# EPICS SNL sequencer program: siteApps/Helium_Inventory-1-0/inventoryApp/src/sncMakeTotalInventory.stt
program sncMakeTotalInventory

option +r;

double massflows[95];
assign massflows to {
	"SCL31-BL01:CM01-LT8401:MassFlow", "SCL31-BL01:CM02-LT8401:MassFlow", "SCL31-BL01:CM03-LT8401:MassFlow", "SCL31-BL01:CM04-LT8401:MassFlow", "SCL31-BL01:CM05-LT8401:MassFlow",
	"SCL31-BL01:CM06-LT8401:MassFlow", "SCL31-BL01:CM07-LT8401:MassFlow", "SCL31-BL01:CM08-LT8401:MassFlow", "SCL31-BL01:CM09-LT8401:MassFlow", "SCL31-BL01:CM10-LT8401:MassFlow",
	"SCL31-BL01:CM11-LT8401:MassFlow", "SCL31-BL01:CM12-LT8401:MassFlow", "SCL31-BL01:CM13-LT8401:MassFlow", "SCL31-BL01:CM14-LT8401:MassFlow", "SCL31-BL01:CM15-LT8401:MassFlow",
	"SCL31-BL01:CM16-LT8401:MassFlow", "SCL31-BL01:CM17-LT8401:MassFlow", "SCL31-BL01:CM18-LT8401:MassFlow", "SCL31-BL01:CM19-LT8401:MassFlow", "SCL31-BL01:CM20-LT8401:MassFlow",
	"SCL31-BL01:CM21-LT8401:MassFlow", "SCL31-BL01:CM22-LT8401:MassFlow", "SCL32-BL02:CM01-LT8401:MassFlow", "SCL32-BL02:CM02-LT8401:MassFlow", "SCL32-BL02:CM03-LT8401:MassFlow",
	"SCL32-BL02:CM04-LT8401:MassFlow", "SCL32-BL02:CM05-LT8401:MassFlow", "SCL32-BL02:CM06-LT8401:MassFlow", "SCL32-BL02:CM07-LT8401:MassFlow", "SCL32-BL02:CM08-LT8401:MassFlow",
	"SCL32-BL02:CM09-LT8401:MassFlow", "SCL32-BL02:CM10-LT8401:MassFlow", "SCL32-BL02:CM11-LT8401:MassFlow", "SCL32-BL02:CM12-LT8401:MassFlow", "SCL32-BL02:CM13-LT8401:MassFlow",
	"P2DT-BL04:CM01-LT8401:MassFlow", "SCL32-BL03:CM01-LT8401:MassFlow", "SCL32-BL03:CM02-LT8401:MassFlow", "SCL32-BL03:CM03-LT8401:MassFlow", "SCL32-BL03:CM04-LT8401:MassFlow",
	"SCL32-BL03:CM05-LT8401:MassFlow", "SCL32-BL03:CM06-LT8401:MassFlow", "SCL32-BL03:CM07-LT8401:MassFlow", "SCL32-BL03:CM08-LT8401:MassFlow", "SCL32-BL03:CM09-LT8401:MassFlow",
	"SCL32-BL03:CM10-LT8401:MassFlow", "SCL32-BL03:CM11-LT8401:MassFlow", "SCL32-BL03:CM12-LT8401:MassFlow", "SCL32-BL03:CM13-LT8401:MassFlow", "SCL32-BL03:CM14-LT8401:MassFlow",
	"SCL32-BL03:CM15-LT8401:MassFlow", "SCL32-BL03:CM16-LT8401:MassFlow", "SCL32-BL03:CM17-LT8401:MassFlow", "SCL32-BL03:CM18-LT8401:MassFlow", "SCL32-BL03:CM19-LT8401:MassFlow",
	"SCL32-BL02:CM01-LT8201:MassFlow", "SCL32-BL02:CM02-LT8201:MassFlow", "SCL32-BL02:CM03-LT8201:MassFlow", "SCL32-BL02:CM04-LT8201:MassFlow", "SCL32-BL02:CM05-LT8201:MassFlow",
	"SCL32-BL02:CM06-LT8201:MassFlow", "SCL32-BL02:CM07-LT8201:MassFlow", "SCL32-BL02:CM08-LT8201:MassFlow", "SCL32-BL02:CM09-LT8201:MassFlow", "SCL32-BL02:CM10-LT8201:MassFlow",
	"SCL32-BL02:CM11-LT8201:MassFlow", "SCL32-BL02:CM12-LT8201:MassFlow", "SCL32-BL02:CM13-LT8201:MassFlow", "P2DT-BL04:CM01-LT8201:MassFlow", "SCL32-BL03:CM01-LT8201:MassFlow",
	"SCL32-BL03:CM02-LT8201:MassFlow", "SCL32-BL03:CM03-LT8201:MassFlow", "SCL32-BL03:CM04-LT8201:MassFlow", "SCL32-BL03:CM05-LT8201:MassFlow", "SCL32-BL03:CM06-LT8201:MassFlow",
	"SCL32-BL03:CM07-LT8201:MassFlow", "SCL32-BL03:CM08-LT8201:MassFlow", "SCL32-BL03:CM09-LT8201:MassFlow", "SCL32-BL03:CM10-LT8201:MassFlow", "SCL32-BL03:CM11-LT8201:MassFlow",
	"SCL32-BL03:CM12-LT8201:MassFlow", "SCL32-BL03:CM13-LT8201:MassFlow", "SCL32-BL03:CM14-LT8201:MassFlow", "SCL32-BL03:CM15-LT8201:MassFlow", "SCL32-BL03:CM16-LT8201:MassFlow",
	"SCL32-BL03:CM17-LT8201:MassFlow", "SCL32-BL03:CM18-LT8201:MassFlow", "SCL32-BL03:CM19-LT8201:MassFlow", "Cryo-CDL00:TBx01-LT8401:2KReturn", "Cryo-CDL00:TBx01-LT8401:2KSupply",
	"Cryo-CDL00:TBx01-LT8401:4KReturn", "Cryo-CDL00:TBx01-LT8401:4KSupply", "Cryo-CDL00:TBx01-LT8401:CDReturn", "Cryo-CDL00:TBx01-LT8401:CDSupply", "Cryo-CDL00:TBx01-LT8401:VLPReturn"
};
monitor massflows;
evflag evWave;
sync massflows evWave;

double	WaveInventory[95];
assign	WaveInventory to "{SYS}{SUBSYS}{DEV}{SUBDEV}Total";
monitor WaveInventory;

int index;
int pvcnt;
ss makewave
{
	state init
	{
		when(TRUE)
		{
		}state MakeWaveInventory
	}

	state MakeWaveInventory
	{
		when(delay(1.) && efTestAndClear(evWave))
		{
			index = 0;
			pvcnt = sizeof(massflows)/sizeof(massflows[0]);
			for(index = 0; index < pvcnt;index++)
			{
				WaveInventory[index]	= massflows[index];
			}
			pvPut(WaveInventory, SYNC);
		}state MakeWaveInventory
	}

}
